{attribute 'GeneratedUsingTerminal: EL2502-0000-0016'}
{attribute addProperty BoxType "EL2502-0000-0016"}
{attribute addProperty Description "EL2502 2Ch. PWM Output, 24V"}
{attribute addProperty Physics "KK"}
{attribute addProperty Id "PWM_Outputs_Channel_1AT %Q*PWM_Outputs_Channel_4C6289CD2PWM_Outputs_Channel_2AT %Q*PWM_Outputs_Channel_4C6289CD2WcStateAT %I*WcState_0B2B16F91InfoDataAT %I*InfoData_32EB74EA10"}
{attribute addProperty CRC "4263597303"}
{attribute addProperty Size "15"}
TYPE EL2502_FE2154F7 EXTENDS EtcSlaveTerminalBase_947E5A46 :
STRUCT
	{attribute addProperty Name "PWM_Outputs_Channel_1"}
	PWM_Outputs_Channel_1 : PWM_Outputs_Channel_4C6289CD;
	{attribute addProperty Name "PWM_Outputs_Channel_2"}
	PWM_Outputs_Channel_2 : PWM_Outputs_Channel_4C6289CD;
	{attribute addProperty Name "WcState"}
	WcState : WcState_0B2B16F9;
	{attribute addProperty Name "InfoData"}
	InfoData : InfoData_32EB74EA;
END_STRUCT
END_TYPE

(* stored: Version 1.2.0.0, ProductVersion 3.1.4024.11
   DUT EL2502_FE2154F7: Id {db262b90-eb19-490a-ae27-ba9533862f17} *)
